# EPICS substitutions: IOCs/12id/iocBoot/ioc12idd/basic_motor.substitutions
file "$(MOTOR)/db/basic_motor.db"
{
pattern
{P,     N,  M,	    DTYP,         C,    S,  DESC,         EGU,      DIR, VELO,  VBAS,  ACCL,  BDST,  BVEL,  BACC,  MRES,   PREC,  DHLM,	DLLM,	INIT}
{12idd:,	1,  "m$(N)",  "OMS VME58",  0,	0,  "motor $(N)", degrees,  Pos, 1,	.1,    .2,    0,     1,	    .2,	   2.5e-4, 5,	  100,	-100,	""}
{12idd:,	2,  "m$(N)",  "OMS VME58",  0,	1,  "motor $(N)", degrees   Pos, 1,	.1,    .2,    0,     1,	    .2,	   2.5e-4, 5,	  100,	-100,	""}
{12idd:,	3,  "m$(N)",  "OMS VME58",  0,	2,  "motor $(N)", degrees   Pos, 1,	.1,    .2,    0,     1,	    .2,	   2.5e-4, 5,	  100,	-100,	""}
{12idd:,	4,  "m$(N)",  "OMS VME58",  0,	3,  "motor $(N)", degrees   Pos, 1,	.1,    .2,    0,     1,	    .2,	   2.5e-4, 5,	  100,	-100,	""}
{12idd:,	5,  "m$(N)",  "OMS VME58",  0,	4,  "motor $(N)", degrees   Pos, 1,	.1,    .2,    0,     1,	    .2,	   2.5e-4, 5,	  100,	-100,	""}
{12idd:,	6,  "m$(N)",  "OMS VME58",  0,	5,  "motor $(N)", degrees   Pos, 1,	.1,    .2,    0,     1,	    .2,	   2.5e-4, 5,	  100,	-100,	""}
{12idd:,	7,  "m$(N)",  "OMS VME58",  0,	6,  "motor $(N)", degrees,  Pos, 1,	.1,    .2,    0,     1,	    .2,	   2.5e-4, 5,	  100,	-100,	""}
{12idd:,	8,  "m$(N)",  "OMS VME58",  0,	7,  "motor $(N)", degrees,  Pos, 1,	.1,    .2,    0,     1,	    .2,	   2.5e-4, 5,	  100,	-100,	""}
}
